INTERFACE I_KeyValueEnumerable EXTENDS __SYSTEM.IQueryInterface

METHOD PUBLIC GetKeyValueEnumerator : I_KeyValueForwardEnumerator
END_METHOD

END_INTERFACE

(* stored: Version 1.1.0.1, ProductVersion 3.1.4024.12
   Itf I_KeyValueEnumerable: Id {20008510-7de6-487c-a47d-e77e9065eb7d}
   Method GetKeyValueEnumerator: Id {4ab6031b-ffe2-4b31-864b-d4e1976557b3} *)
